// Annex B — cylinder HAL: 2 outputs, 2 position sensors
TYPE ST_CylinderHal :
STRUCT
    ExtendOut, RetractOut   : BOOL;
    ExtendedFb, RetractedFb : BOOL;
END_STRUCT
END_TYPE

(* stored: Version 1.1.0.1, ProductVersion 3.1.4024.12
   DUT ST_CylinderHal: Id {ec131bff-ed04-4aa1-9364-5aa7cc7c9466} *)
